PROGRAM MAIN
VAR
END_VAR

LadderLogicBottleChecker();

END_PROGRAM

(* stored: Version 1.1.0.1, ProductVersion 3.1.4026.8
   POU MAIN: Id {2167deda-e464-40be-b535-575ae174f84c}, SpecialFunc None *)
